(* IEC 61131-3 sources: traffic-lights/PLC_TrafficLights/Class/Road, 1 file *)

(* ---- Road.st ---- *)
(*!
<Class
	Name               = "Road"
	Revision           = "0.0"
	RealtimeTask       = "false"
	CyclicTask         = "true"
	DefCyclictime      = "100 ms"
	BackgroundTask     = "false"
	Sigmatek           = "false"
	OSInterface        = "false"
	HighPriority       = "false"
	Automatic          = "false"
	UpdateMode         = "Prescan"
	SharedCommandTable = "true"
	Objectsize         = "(752,120)">
	<Channels>
		<Server Name="ClassSvr" Visualized="false" Initialize="false" WriteProtected="true" Retentive="false"/>
		<Server Name="Svr_AverageWaitingTime" Visualized="true" Initialize="false" WriteProtected="true" Retentive="false"/>
		<Server Name="Svr_IncomingCars" Visualized="true" Initialize="false" WriteProtected="false" Retentive="false"/>
		<Server Name="Svr_PassingTime" Visualized="false" Initialize="true" DefValue="1200" WriteProtected="false" Retentive="SRam"/>
		<Server Name="Svr_TotalCarsPassed" Visualized="true" Initialize="false" WriteProtected="true" Retentive="false"/>
		<Client Name="I_TrafficLight" Required="false" Internal="false"/>
	</Channels>
	<RevDoku>
		<Owner Company="Eqraft"/>
		<Dokumentation Revision="0.1.0" Date="2024-06-20" Author="Klaas Post" Company="Eqraft"/>
	</RevDoku>
</Class>
*)
Road : CLASS
  //Servers:
	ClassSvr 	: SvrChCmd_DINT;
	Svr_IncomingCars 	: SvrCh_DINT;
	Svr_TotalCarsPassed 	: SvrCh_DINT;
	Svr_AverageWaitingTime 	: SvrCh_REAL;
	Svr_PassingTime 	: SvrCh_UDINT;
  //Clients:
	I_TrafficLight 	: CltCh__LightColor_PTofCls_TrafficLight;
  //Variables:
		tLastCarPassed 	: UDINT;
		TotalWaitingTime 	: UDINT;
  //Functions:

	FUNCTION VIRTUAL GLOBAL CyWork
		VAR_INPUT
			EAX 	: UDINT;
		END_VAR
		VAR_OUTPUT
			state (EAX) 	: UDINT;
		END_VAR;
  //Tables:
	FUNCTION @STD
		VAR_OUTPUT
			ret_code	: CONFSTATES;
		END_VAR;
	FUNCTION GLOBAL TAB @CT_;
END_CLASS;

//----------------------------------------------------------------------------------------------------
//  Standard class methods
//----------------------------------------------------------------------------------------------------

// Standard Cywork, runs every set amount of time.
FUNCTION VIRTUAL GLOBAL Road::CyWork
	VAR_INPUT
		EAX 	: UDINT;
	END_VAR
	VAR_OUTPUT
		state (EAX) 	: UDINT;
	END_VAR

    IF OPS.tAbsolute - tLastCarPassed > Svr_PassingTime THEN

        // If there's no cars waiting, exit function.
        IF Svr_IncomingCars < 1 THEN
            state := READY;
            RETURN;
        END_IF;

        // Car(s) read the traffic light.
        I_TrafficLight := I_TrafficLight.Read();

        // If the signal is red, exit function.
        IF I_TrafficLight = TrafficLight::eRed THEN
            TotalWaitingTime += Svr_PassingTime;
            state := READY;
            RETURN;
        END_IF;

        // If light is yellow, traffic might pass or might not.
        IF I_TrafficLight = TrafficLight::eYellow & OPS.tAbsolute MOD 5 = 0 THEN
            TotalWaitingTime += Svr_PassingTime;
            RETURN;
        END_IF;

        // Car is free to go so decrease incoming traffic by one and add to total of cars passed.
        Svr_IncomingCars -= 1;
        Svr_TotalCarsPassed += 1;

        tLastCarPassed := OPS.tAbsolute;
    END_IF;

    IF Svr_TotalCarsPassed > 0 THEN
        Svr_AverageWaitingTime := TotalWaitingTime / Svr_TotalCarsPassed;
    ELSE
        Svr_AverageWaitingTime := 0;
    END_IF;

	state := READY;

END_FUNCTION
